SUBAPPLICATION Tuple (* Subapplication Type *)
  (* Standard: 61499-2 *)
  (* Version 1.0, 2023-02-17, Franz *)
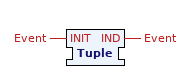
  EVENT_INPUT
    INIT;
  END_EVENT
  EVENT_OUTPUT
    IND;
  END_EVENT
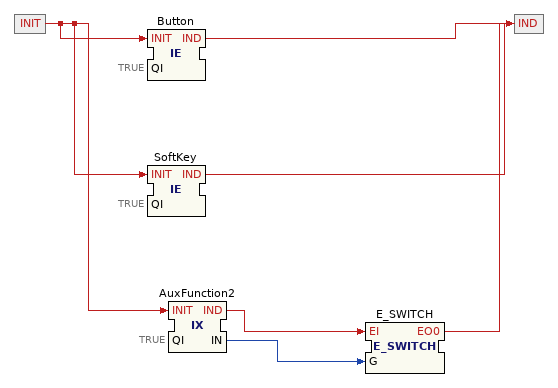
  FBS
    Button : IE(QI := TRUE);
    SoftKey : IE(QI := TRUE);
    AuxFunction2 : IX(QI := TRUE);
    E_SWITCH : E_SWITCH;
  END_FBS
  EVENT_CONNECTIONS
    INIT TO Button.INIT;
    Button.IND TO IND;
    INIT TO SoftKey.INIT;
    SoftKey.IND TO IND;
    INIT TO AuxFunction2.INIT;
    AuxFunction2.IND TO E_SWITCH.EI;
    E_SWITCH.EO0 TO IND;
  END_CONNECTIONS
  DATA_CONNECTIONS
    AuxFunction2.IN TO E_SWITCH.G;
  END_CONNECTIONS
END_SUBAPPLICATION
